FUNCTION_BLOCK FB_937A_VG
VAR_IN_OUT
	VG : ST_VG;
END_VAR
VAR_INPUT
	PG	:	ST_VG := g_DummyVG;
END_VAR
VAR_OUTPUT
END_VAR
VAR
	rV	:	LREAL;
END_VAR

(* 937A Logarithmic Output Conversion *)
(* 7-15-2015 *)
(* This function will read the pressure from any gauge on a 937A. *)

rV := LREAL#10*INT_TO_LREAL(VG.iPRESS_R)/LREAL#32767;
VG.rPRESS := LREAL_TO_REAL(EXPT(10,rV/LREAL#0.6-LREAL#12));


(* Ion Gauge Protection Functions *)
(* If the PG pressure is greater than the VG.PRO_SP then the gauge is disabled *)
(* If the PG pressure is less than the VG.PRO_SP then the gauge is enabled *)
(* This FB also implements some hysteresis so the gauge doesn't have rapid power cycling while near the turn on boundary *)

IF PG.rPRESS < VG.rPRO_SP THEN

VG.xHV_DIS := NOT VG.xHV_SW;

ELSIF NOT VG.xHV_DIS THEN
	IF VG.rPRESS > VG.rPRO_SP + VG.rHYS_PR OR PG.rPRESS > VG.rPRO_SP + VG.rHYS_PR THEN
		VG.xHV_DIS := TRUE;
	END_IF
ELSE
	VG.xHV_DIS := TRUE;
END_IF


(* Pressure gauge OK checks *)
VG.xPRESS_OK := (rV <=9.6 ) AND (rV>=0.6); //legacy

IF (rV <=9.6 ) AND (rV>=0.6) THEN
	VG.eState := E_PressureState.Valid; // normal
ELSIF rV >= 0.18 AND rV <= 0.22 THEN
	VG.eState := E_PressureState.ValidLo; //LO
ELSIF rV >= 9.7 AND rV<= 9.9 THEN
	VG.eState := E_PressureState.ValidHi; //HIGH
ELSIF rV < 0.18 THEN
	VG.eState := E_PressureState.GaugeDisconnected; //not on
ELSE
	VG.eState := E_PressureState.PressInvalid; //other fault - could be no gauge, controller powering up etc
END_IF

(* Setpoint evaluation *)
VG.xAT_VAC := (VG.eState = E_PressureState.Valid) AND VG.rPRESS < VG.rVAC_SP;

END_FUNCTION_BLOCK

(* stored: Version 1.1.0.1, ProductVersion 3.1.4022.10
   POU FB_937A_VG: Id {0483146b-b0e8-4c2d-b90b-7317630633a1}, SpecialFunc None *)
